// TIA Portal V19 export
FUNCTION_BLOCK "DriveInterface"   // FB7, LAD
TITLE = Drive Interface
// stored: Access Published, MemoryReserve 100, SetENOAutomatically false
   VAR_INPUT
      PowerRequest : Bool;
      Reset : Bool;
      Run : Bool;
   END_VAR
   VAR_OUTPUT
      DrivePower : Bool;
      DriveReset : Bool;
      DriveRun : Bool;
   END_VAR
   VAR
      TOF_Power : IEC_TIMER;
      TOF_Reset : IEC_TIMER;
   END_VAR
BEGIN

REGION Network 1: Drive Power
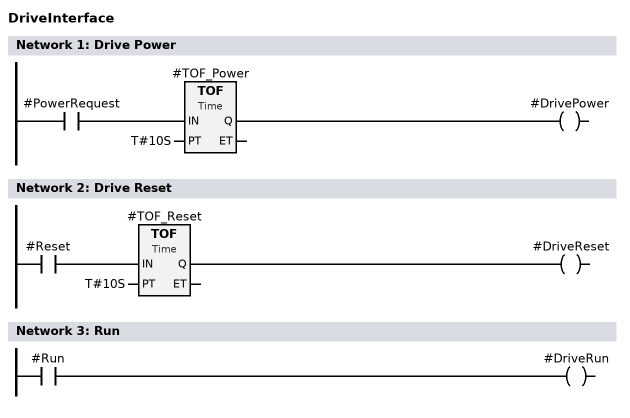
   RUNG wire#powerrail
      Contact( #PowerRequest )
      { S7_Templates := "time_type := Time" } #TOF_Power.TOF(pt := T#10S, et =>)
      Coil( #DrivePower )
   END_RUNG
   // the same network as SCL:
   #TOF_Power.TOF(IN := #PowerRequest, PT := T#10S);
   #DrivePower := #TOF_Power.Q;
END_REGION

REGION Network 2: Drive Reset
   RUNG wire#powerrail
      Contact( #Reset )
      { S7_Templates := "time_type := Time" } #TOF_Reset.TOF(pt := T#10S, et =>)
      Coil( #DriveReset )
   END_RUNG
   // the same network as SCL:
   #TOF_Reset.TOF(IN := #Reset, PT := T#10S);
   #DriveReset := #TOF_Reset.Q;
END_REGION

REGION Network 3: Run
   RUNG wire#powerrail
      Contact( #Run )
      Coil( #DriveRun )
   END_RUNG
   // the same network as SCL:
   #DriveRun := #Run;
END_REGION
END_FUNCTION_BLOCK
